GLOBALCONSTANTS Hutschienenmoped_XL_LED_COLOURS (* Global constants *)
  (* Standard: 61499-1 *)
  (* Version 1.0, 2024-01-25, franz *)
  VAR_GLOBAL CONSTANT
    LED_GREEN : UINT := 1;
    LED_BLUE : UINT := 2;
    LED_RED : UINT := 3;
    LED_WHITE : UINT := 4;
    LED_BLACK : UINT := 5;
    LED_MAGENTA : UINT := 6;
    LED_CYAN : UINT := 7;
    LED_YELLOW : UINT := 8;
  END_VAR
END_GLOBALCONSTANTS
